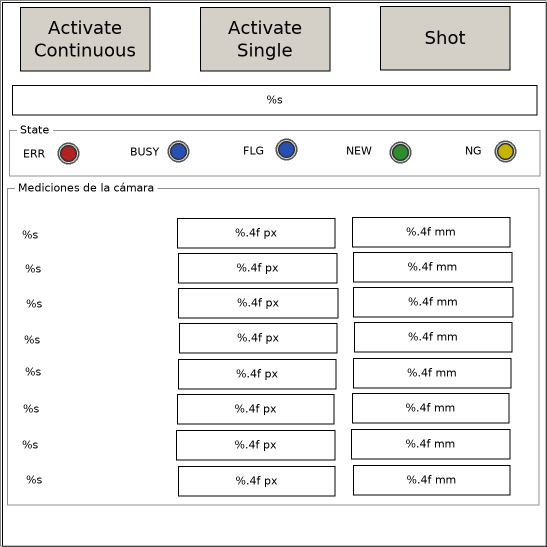
VISUALIZATION VisionHMI  // 547x547
    Rectangle (2,2 545x545)
    Rectangle (200,7 130x64), "Activate Single"
        toggle HMI.Bt_ActivateSingle
    Rectangle (12,85 525x30), "%s", text variable: GVL.Vision.State
    Rectangle (380,6 130x64), "Shot"
        tap HMI.Bt_Shot
    GroupBox (7,180 532x325), "Mediciones de la cámara"
        Rectangle (170,38 158x30), "%.4f px", text variable: GVL.VisionResults[0]
        Rectangle (171,73 159x30), "%.4f px", text variable: GVL.VisionResults[1]
        Rectangle (171,108 160x30), "%.4f px", text variable: GVL.VisionResults[2]
        Rectangle (172,143 158x30), "%.4f px", text variable: GVL.VisionResults[3]
        Rectangle (171,179 158x30), "%.4f px", text variable: GVL.VisionResults[4]
        Rectangle (170,214 157x30), "%.4f px", text variable: GVL.VisionResults[5]
        Rectangle (169,250 159x30), "%.4f px", text variable: GVL.VisionResults[6]
        Rectangle (171,286 157x30), "%.4f px", text variable: GVL.VisionResults[7]
        Rectangle (345,37 158x30), "%.4f mm", text variable: GVL.VisionResultsmm[0]
        Rectangle (12,40 150x30), "%s", text variable: HMI.MeasurementNames[0]
        Rectangle (15,74 150x30), "%s", text variable: HMI.MeasurementNames[1]
        Rectangle (16,109 150x30), "%s", text variable: HMI.MeasurementNames[2]
        Rectangle (14,145 150x30), "%s", text variable: HMI.MeasurementNames[3]
        Rectangle (15,177 150x30), "%s", text variable: HMI.MeasurementNames[4]
        Rectangle (13,214 150x30), "%s", text variable: HMI.MeasurementNames[5]
        Rectangle (12,250 150x30), "%s", text variable: HMI.MeasurementNames[6]
        Rectangle (16,285 150x30), "%s", text variable: HMI.MeasurementNames[7]
    Rectangle (20,7 130x64), "Activate Continuous"
        toggle HMI.Bt_ActivateContinuous
    GroupBox (9,122 531x54), "State"
        Label (11,17 32x30), "ERR"
        Lamp1 (45,19 29x25), variable: GVL.Vision.SensorToPlc.ERR, style: Lamp-Lamp1-Red
        Label (118,15 38x30), "BUSY"
        Lamp1 (155,17 29x25), variable: GVL.Vision.SensorToPlc.BUSY, style: Lamp-Lamp1-Blue
        Label (231,14 38x30), "FLG"
        Lamp1 (263,15 29x25), variable: GVL.Vision.SensorToPlc.FLG, style: Lamp-Lamp1-Blue
        Label (334,14 38x30), "NEW"
        Lamp1 (377,18 29x25), variable: HMI.L_NewMeasurement, style: Lamp-Lamp1-Green
        Label (453,14 38x30), "NG"
        Lamp1 (482,17 29x25), variable: GVL.Vision.SensorToPlc.OR_Jud, style: Lamp-Lamp1-Yellow
    Rectangle (353,252 159x30), "%.4f mm", text variable: GVL.VisionResultsmm[1]
    Rectangle (353,287 160x30), "%.4f mm", text variable: GVL.VisionResultsmm[2]
    Rectangle (354,322 158x30), "%.4f mm", text variable: GVL.VisionResultsmm[3]
    Rectangle (353,358 158x30), "%.4f mm", text variable: GVL.VisionResultsmm[4]
    Rectangle (352,393 157x30), "%.4f mm", text variable: GVL.VisionResultsmm[5]
    Rectangle (351,429 159x30), "%.4f mm", text variable: GVL.VisionResultsmm[6]
    Rectangle (353,465 157x30), "%.4f mm", text variable: GVL.VisionResultsmm[7]
END_VISUALIZATION

(* stored: Version 1.1.0.1, ProductVersion 3.1.4024.9
   Visu VisionHMI: Id {161fa826-06c7-472c-a227-5c70174cba46} *)
